ABB RAPID module: CalibData.modx

MODULE CalibData
    PERS tooldata Front_TCP:=[TRUE,[[130.508928334,-200,71.951905284],[1,0,0,0]],[1,[0,0,0.001],[1,0,0,0],0,0,0]];
    PERS tooldata Pen_TCP:=[TRUE,[[4.330131423,2.499983828,300.00000007],[1,0,0,0]],[1,[0,0,0.001],[1,0,0,0],0,0,0]];
    PERS tooldata Back_TCP :=[TRUE,[[-14.565,0,98.4],[0.707107,0,0.707107,0]],[1.5,[0,0,66.18],[1,0,0,0],0,0,0]];
ENDMODULE
